// TwinCAT 3 PLC project Main
// ProgramVersion: 3.1.4023.0
// libraries:
//   Tc2_Standard, * (Beckhoff Automation GmbH)
//   Tc2_System, * (Beckhoff Automation GmbH)
//   Tc2_Utilities, * (Beckhoff Automation GmbH)
//   Tc3_Module, * (Beckhoff Automation GmbH)
// project tree:
//   / PlcTask.TcTTO
//   POUs/ MAIN.TcPOU
// real-time tasks:
//   TASK PlcTask: cycle T#10ms, priority 20, ADS port 350

CONFIGURATION Main
    RESOURCE PLC ON TwinCAT3
        TASK PlcTask(INTERVAL := T#10ms, PRIORITY := 20);
        PROGRAM MAIN WITH PlcTask : MAIN;
    END_RESOURCE
END_CONFIGURATION

// ---- POUs/MAIN.TcPOU
PROGRAM MAIN
VAR

	start 		:BOOL;
	ip			:STRING := '127.0.0.1'; // is the address which will be pinged.
	pingReply 	:INT := -1; // -1 for pending, 0 for ping failed, 1 ping succeeded
	
	comndLine	:STRING(139);
	ping 		:NT_StartProcess;

END_VAR

// You will need to run the following commands on your IPC using Administrator Powershell. 
// This is to install the TcXaeMgmt package in powershell which the below command will use.
// ----------------------------------------------------------------------------------------
// Set-ExecutionPolicy -ExecutionPolicy RemoteSigned
// Exit
// ----------------------------------------------------------------------------------------
// Now run the file bellow as administrator.
// .\\Modules\TcXaeMgmt\install.bat 
// ----------------------------------------------------------------------------------------
// You can check if this worked by verifying if the folder bellow exist and has content.
// C:\Program Files\WindowsPowerShell\Modules\TcXaeMgmt\3.2.25

// To use
// ------
// Main.pingReply is used for the feedback
// set start to true to run a ping test. 
// approximately 5 seconds to have a ping succeeded result. 
// approximately 10 seconds to have a ping failed result. 

comndLine:=CONCAT(STR1:='""""Main.pingReply"""" -value (Test-Connection -ComputerName ', STR2:=ip);
comndLine:=CONCAT(STR1:=comndLine, STR2:=' -Quiet) -Force;Close-TcSession -InputObject $$s;"", 0: window.close")');

ping(
	NetId := '',
	PathStr := 'C:\Windows\System32\mshta vbscript:Execute("CreateObject(""WScript.Shell"").Run ""powershell -c $$r=get-adsroute -local;$$s=New-TcSession -Route $$r -Port 851;Write-TcValue -Session $$s -Path ',
	DirName := 'C:\Windows\System32',
	ComndLine := comndLine,
	Start := start,
	TmOut := DEFAULT_ADS_TIMEOUT
);

IF start THEN
	pingReply := -1;
	start := FALSE;
END_IF

END_PROGRAM
